# EPICS substitutions: maglps/Db/maglpsCPU.substitutions
global {PLC=PLCCPU, HOLDHIGH=1.0}

file "maglpsConn.template"
{
	pattern {SGNL}
		{CPU}
}

file "maglpsCPUR.template"
{
	pattern {SGNL, SOFF}
		{CPU, 0}
}

file "maglpsCPUInternal.template"
{
	pattern {SGNL}
		{CPU}
}

file "maglpsCPUW.template"
{
	pattern {SGNL, SOFF}
		{CPU, 0}
}
